# B&R Automation Studio project Nitto (part 2)

### Global.typ - Global data types
```iecst
(********************************************************************
 * COPYRIGHT -- Bernecker + Rainer
 ********************************************************************
 * File: Global.typ
 * Author: schoenefeldr
 * Created: July 06, 2012
 ********************************************************************
 * Global data types of project 120706_hp_001
 ********************************************************************)
(*======================================================================================================================================*)
(*GLOBAL OPERATING MODE DEFINITIONS*)
(*======================================================================================================================================*)
(*General operating mode of the machine*)

TYPE
	OpModeEnum_Type :
		(
		OPMODE_MANUAL := 0, (*Manual mode ("Hand")*)
		OPMODE_AUTOMATIC := 1, (*Automatic mode*)
		OPMODE_SETUP := 2, (*Automatic mode with additional functions ("Einrichten")*)
		OPMODE_SERVICE := 5 (*Service mode with direct access to hardware*)
		);
END_TYPE

(*General machine status*)

TYPE
	MachineStatusEnum_Type :
		(
		STATE_PREOPERATIONAL := 0, (*Machine not ready for operation*)
		STATE_READY_FOR_OPERATION := 1, (*Machine ready for operation*)
		STATE_AUTOMATIC := 2, (*Machine is running in operating mode automatic*)
		STATE_JOG := 3, (*Jog mode active*)
		STATE_MANUAL := 4, (*Manual operating mode*)
		STATE_FAULT := 5 (*Fault active*)
		);
END_TYPE

(*Cutting unit operating mode*)

TYPE
	OpModeCutEnum_Type :
		(
		CUT_DISABLED := 20, (*Cut unit disabled*)
		FREE_CUT := 21, (*Free cutting mode*)
		PHYSICAL_TRIGGER := 22, (*synchronous cutting mode*)
		VIRTUAL_TRIGGER := 23 (*synchronous cutting mode*)
		);
END_TYPE

(*Laaminator operating mode 17.01.14 opirational Mode*)

TYPE
	OpModeLaminatorEnum_Type :
		(
		LAMINATOR_DISABLED := 0,
		LAMINATOR_ENABLED := 1
		);
END_TYPE

(*Label dispenser operating mode*)

TYPE
	OpModeLabelDispenser_Type :
		(
		LABEL_DISP_DISABLED := 0, (*Label dispenser disabled*)
		LABEL_DISP_ENABLED := 1 (*Label dispenser enabled*)
		);
END_TYPE

(*Long cut unit operating mode*)

TYPE
	OpModeLongCutEnum_Type :
		(
		LONG_CUT_DISABLED := 10, (*Long cut enabled*)
		LONG_CUT_ENABLED := 11 (*active braking*)
		);
END_TYPE

(*Winder operating mode*)

TYPE
	OpModeWinderEnum_Type :
		(
		WIND_DISABLED := 35, (*Winder disabled*)
		WINDER := 36, (*Machine ready for operation*)
		BRAKE := 37 (*Brake functionality*)
		);
END_TYPE

(*Web tension unit operating mode*)

TYPE
	OpModeTensionEnum_Type :
		(
		WEB_TENSION_DISABLED := 5, (*Web tension control disabled*)
		WEB_TENSION_ENABLED := 6 (*Web tension control enabled*)
		);
END_TYPE

(*End module operating mode*)

TYPE
	OpModeEndModuleEnum_Type :
		(
		END_MODULE_DISABLED := 40, (*No end module selected, disable winder and belts*)
		END_MODULE_TOP_WINDER := 41, (*Select top winder*)
		END_MODULE_BOT_WINDER := 42, (*Select bottom winder*)
		END_MODULE_TANDEM_WINDER := 43, (*Select tandem winder*)
		END_MODULE_BELTS := 44 (*Select upper belt and conveyor belt*)
		);
END_TYPE

(*Markpoint operating mode*)

TYPE
	OpModeMarkpointEnum_Type :
		(
		DISABLED := 0, (*deactivated*)
		SENSOR_CONTROL := 1, (*Use sensor*)
		PERIOD_CONTROL := 2 (*use period*)
		);
	CONST_MACHINE_MODES_Type : 	STRUCT
		MANUAL : INT := 0;
		AUTOMATIC : INT := 1;
		PRODUCTION : INT := 2;
		SAFETYSTOP : INT := 7;
		RESET : INT := 8;
		EMERGENCYSTOP : INT := 9;
	END_STRUCT;
END_TYPE

(*Machine structure*)

TYPE
	Machine_Type : 	STRUCT
		Command : MachineCmd_Type;
		Safety : MachineSafe_Type;
		Data : MachineData_Type;
		Config : MachineCfg_Type;
		IO : MachineIo_Type; (*Inputs on DI9371-38A7 to DI9371-38A10*)
		Status : MachineStatus_Type;
	END_STRUCT;
	MachineCmd_Type : 	STRUCT
		StartRequestButton : BOOL; (*Start request by pressing of button*)
		StopRequestButton : BOOL; (*Stop request by pressing of button*)
		AutoStopRequestAlarm : BOOL; (*Stop request by alarm handling (automatic mode only)*)
		JogRequestButton : BOOL; (*Jog request by pressing of button*)
		UpdateRecipe : BOOL; (*Command for updating recipe parameters*)
		OpModeSet : OpModeEnum_Type; (*operating mode setpoint*)
		MasterVelocity : REAL; (*master velocity setpoint [µm/s]*)
	END_STRUCT;
	MachineSafe_Type : 	STRUCT
		RequestSTO : BOOL; (*Emergency Stop is requested (active low)*)
		RequestSLS : BOOL; (*Safe Limited Speed requested by opening safety doors (active low)*)
		ResetSafeMC : BOOL; (*Reset input of SafeMC Function Blocks*)
		ResetStartupInhibit : BOOL; (*Reset emergency functions (quit startup inhibit)*)
		ResetUserSafeMC : BOOL;
		SLSmasterVeloScaled : REAL; (*maximum master velocity command if SLS is requested due to scalings of cutting units*)
	END_STRUCT;
	MachineData_Type : 	STRUCT
		cut1 : MachineDataCut_Type; (*Derived data for cutting unit 1*)
		cut2 : MachineDataCut_Type; (*Derived data for cutting unit 2*)
		AccMaster : BOOL; (*Accelerate master axis*)
		StopMaster : BOOL; (*Decelerate master axis with machine deceleration ramp*)
		DiscreteMove : BOOL; (*Discrete move over distance or fixed number of packages*)
		VelocityIncrement : REAL; (*Increment for accelerate / decelerate master*)
	END_STRUCT;
	MachineDataCut_Type : 	STRUCT  (*Derived cuttin unit data *)
		cutPeriodLength : REAL; (*Material period corresponding to cutting cylinder perimeter [µm]*)
		scaleCutToMasterPeriod : REAL; (*Scaling factor for conversion of cutting unit into master unit*)
	END_STRUCT;
	MachineCfg_Type : 	STRUCT  (*Configuration data structure*)
		FlengeDMS : USINT; (*Configuration of Flenge DMS analogue input*)
	END_STRUCT;
	MachineStatus_Type : 	STRUCT
		initDone : BOOL; (*Initialisation complete*)
		recipeUpdating : BOOL; (*recipe updating is active*)
		recipeUpdateDone : BOOL; (*recipe update in all units completed*)
		Diam : MachineStatusDiam_Type; (*actual diameters*)
		Act : MachineStatusEnum_Type; (*actual machine status*)
		OpModeAct : OpModeEnum_Type; (*actual operating mode*)
		CalcDiam : MachineCalcDiam_Type; (*actual estimated diameter *)
		Power : BOOL; (*drives enabled*)
		ReferencedOK : BOOL; (*Combination of necessary reference conditions to start*)
		SupportSpikesOK : BOOL; (*Necessary supportspikes for tandem winders are closed*)
		mManualModeActive : BOOL;
		mAutoModeActive : BOOL;
		StartButtonBlinking : BOOL;
		StartButtonActOut : BOOL;
		WebBreakLabeler : BOOL;
		EnableMasterMove : BOOL;
	END_STRUCT;
	MachineStatusDiam_Type : 	STRUCT
		MainUnwind : REAL; (*Actual diameter Abwicklung*)
		Spend1 : REAL; (*Actual diameter Abwickler 1*)
		Spend2 : REAL; (*Actual diameter Abwickler 2*)
		Spend3 : REAL; (*Actual diameter Abwickler 3*)
		Spend4 : REAL; (*Actual diameter Abwickler 4*)
		Grid1 : REAL; (*Actual diameter Gitteraufwickler 1*)
		Grid2 : REAL; (*Actual diameter Gitteraufwickler 2*)
		Laminator1 : REAL; (*Actual diameter Laminator 1*)
		Laminator2 : REAL; (*Actual diameter Laminator 2*)
		TUnwindTop : REAL; (*Actual diameter Tandemwickler oben*)
		TUnwindBot : REAL; (*Actual diameter Tandemwickler unten*)
	END_STRUCT;
	MachineCalcDiam_Type : 	STRUCT
		MainUnwind : REAL; (*Actual estimated diameter Abwicklung*)
		TUnwindTop : REAL; (*Actual estimated diameter Tandemwickler oben*)
		TUnwindBot : REAL; (*Actual estimated diameter Tandemwickler unten*)
	END_STRUCT;
END_TYPE

(*Data types for print marks*)

TYPE
	PrintMark_Type : 	STRUCT
		Data : PrintMarkData_Type;
		ActIndex : USINT;
		MaxArrIndex : USINT;
	END_STRUCT;
	PrintMarkData_Type : 	STRUCT
		ActDiff : REAL;
		LastPos : REAL;
		AbsPos : REAL;
	END_STRUCT;
END_TYPE

(*Data types for visualisation*)

TYPE
	Visu_Type : 	STRUCT
		RelSafeOut : BOOL;
		Cmd : VisuCmd_Type;
		Status : VisuStatus_Type;
	END_STRUCT;
	VisuCmd_Type : 	STRUCT
		pageSel : VisuCmdPage_Type;
		resetError : BOOL;
		DoReference : BOOL;
		Hold : BOOL;
		StartAddPos : BOOL;
		numPkg : UDINT; (*Input for movement over a number of packages*)
		jogOverride : REAL; (*override for jogging in percent*)
		masterPos : REAL;
		masterVelo : REAL;
	END_STRUCT;
	VisuCmdPage_Type : 	STRUCT
		selPage : UINT;
		reqPage : UINT;
		actPage : UINT := 100;
		newPage : UINT;
		oldPage : UINT;
	END_STRUCT;
	VisuStatus_Type : 	STRUCT
		ActVelocity : REAL; (*Actual master speed [µm/s]*)
		ActPosition : REAL; (*Actual master position [µm]*)
	END_STRUCT;
	mAutoPunchPar_typ : 	STRUCT
		Mode : OpModeCutEnum_Type;
		TriggerIndex : USINT;
		RmWindow : REAL;
		PositionPunch : DINT;
		PositionSensor : DINT;
		CutStartPos : DINT;
		CutEndPos : DINT;
		Insetting : REAL;
		RegMarkPosition : DINT;
		MaxCorr : DINT;
	END_STRUCT;
		RmIfStatusActVal_Type : 	STRUCT  (*Structure for actual data, positions, differences etc.*)
		RmDetected : BOOL; (*A registration mark has been detected during the last movement*)
		RmShiftValid : BOOL; (*The shift value has been calculated after a valid registration mark has been detected*)
		lastValidIndex : USINT; (*Returns the last valid index of the RM data*)
		RegMark : ARRAY[0..MAX_RM_DATA_ARRAY_INDEX]OF RmActValArray_Type; (*Arrays for each registraion mark sensor*)
	END_STRUCT;
		RmActValArray_Type : 	STRUCT  (*Structure for actual data for visualisation*)
		Ident : UDINT; (*Serial number of the registration mark*)
		PIdx : USINT; (*Group index for this RM*)
		RegMarkActPos : DINT; (*Actual RM position [axis units]*)
		AbsPosition : REAL; (*Absolute position of the RM [µm]*)
		Difference : REAL; (*Difference between absolute positions [µm]*)
		SetpointError : REAL; (*Difference between RM position and setpoint [µm]*)
	END_STRUCT;
		reg_mark_typ : 	STRUCT  (*control structure*)
		Command : reg_mark_command_typ; (*command structure*)
		Parameter : reg_mark_parameter_typ; (*parameter structure*)
		Data : reg_mark_data_typ; (*data structure*)
		Status : reg_mark_status_typ; (*status structure*)
	END_STRUCT;
		reg_mark_command_typ : 	STRUCT  (*command structure*)
		StartCorrection : BOOL; (*start the correction*)
		StopCorrection : BOOL; (*stop the correction*)
		SearchTrigger : BOOL; (*search trigger manual*)
		ResetCalc : BOOL; (*reset the calculation data*)
		InitCalcData : BOOL; (*initialize the changed calculation parameters*)
		InitCaptureData : BOOL; (*initialize the changed capture parameters *)
	END_STRUCT;
	reg_mark_parameter_typ : 	STRUCT  (*parameter structure*)
		Mode : USINT; (*RM control mode, e.g. real RMs, virtual RMs etc.*)
		RegMarkAdditiveSetpoint : REAL; (*Additive cumulated RM position*)
		Capture : reg_mark_parameter_capture_typ; (*capture parameter structure*)
		Calculation : MC_RMCALC001_REF; (*ControllerParameter input structure of MC_BR_RegMarkCalc001*)
		Shift : reg_mark_parameter_shift_typ; (*shift parameter structure*)
	END_STRUCT;
	reg_mark_parameter_capture_typ : 	STRUCT  (*capture parameter structure*)
		Trigger : MC_BR_TRIGGER_REF; (*trigger input structure of MC_BR_RegMarkCapture001*)
		Product : MC_BR_PRODUCT_REF; (*product input structure of MC_BR_RegMarkCapture001*)
		WindowNegative : REAL; (*window in which the valid trigger signal can occur before the expected position*)
		WindowPositive : REAL; (*window in which the valid trigger signal can occur after the expected position*)
		DistanceToSensor : REAL; (*distance between the sensor and the cut/seal position*)
	END_STRUCT;
	reg_mark_parameter_shift_typ : 	STRUCT  (*shift parameter structure*)
		Velocity : REAL; (*maximum velocity for reaching the shift *)
		Acceleration : REAL; (*maximum acceleration for reaching the shift*)
		ApplicationDistanceRatio : REAL; (*ratio of shift application distance / product length (must be <1.0!!!)*)
	END_STRUCT;
	reg_mark_data_typ : 	STRUCT
		resetDone : BOOL; (*handshake with interface for reset command*)
		probeTriggered : BOOL; (*handshake with touchProbe*)
		actRmArrIndex : USINT; (*Write pointer index for array of RM data*)
		axisIndex : USINT; (*Index on global axis handle*)
		config : UDINT; (*configuration bits (available etc.)*)
		attrib : UDINT; (*attribute bits (reserved)*)
		rmStep : USINT; (*general registration mark control step state*)
		tpStep : USINT; (*touch probe step state*)
		lastNumOfValidTriggers : UDINT; (*Last number of valid triggers*)
		receiveParID : UINT; (*ParID of the cyclic data transfer-channel that has been automatically determined*)
		eventDelayTime : REAL; (*estimated transmission delay time [s] (unit "s" avoids division in cyclic task)*)
		eventDelayPosCompensation : REAL; (*estimated position correction for compensation of transmission delay via POWERLINK*)
	END_STRUCT;
	reg_mark_status_typ : 	STRUCT  (*status structure*)
		initDone : BOOL; (*Initialisation completed*)
		Capture : reg_mark_status_capture_typ; (*capture status structure*)
		Calculation : reg_mark_status_calc_typ; (*calculation status structure*)
		ErrorID : UINT; (*ErrorID if an function block reports an error*)
	END_STRUCT;
	reg_mark_status_capture_typ : 	STRUCT  (*capture status structure*)
		ValidTriggers : UDINT; (*number of valid triggers found by the function block*)
		MissedTriggers : UINT; (*number of missed triggers*)
		ActProbePosition : DINT; (*actual position of the last found trigger by TouchProbe*)
		ActLength : REAL; (*actual length of the last found trigger*)
		ActLengthIV : REAL; (*actual length of the interval*)
		ActPosition : REAL; (*actual position of the last found trigger*)
		LengthError : REAL; (*length error of the last interval*)
		SavePositionError : REAL; (*save variable for change detection*)
		PositionError : REAL; (*actual position error of the last found trigger*)
		SetpointError : REAL; (*Setpoint error between RM position setpoint and RM position actual value [µm]*)
		Reserve : REAL; (*Reserve*)
	END_STRUCT;
	reg_mark_status_calc_typ : 	STRUCT  (*calculation status structure*)
		ErrorID : UINT; (*ErrorID*)
		ValidCorrections : UDINT; (*number of valid calculated corrections*)
		Distance : REAL; (*calculated distance difference*)
		Shift : REAL; (*calculated shift*)
		DistanceLimiterActive : BOOL; (*shows if the calculated distance was limited to maximum*)
		ShiftLimiterActive : BOOL; (*shows if the calculated shift was limited to maximum*)
	END_STRUCT;
		RmIf_Type : 	STRUCT
		Command : RmIfCmd_Type; (*Command structure*)
		Para : RmIfPara_Type; (*Parameter structure*)
		Data : RmIfData_Type; (*General data structure*)
		Status : RmIfStatus_Type; (*Status structure*)
		Error : RmIfError_Type; (*Error data structure*)
	END_STRUCT;
	RmIfCmd_Type : 	STRUCT  (*Command structure*)
		startGeneral : BOOL; (*command for starting (depends on operating mode)*)
		stopGeneral : BOOL; (*command for starting (depends on operating mode)*)
		updatePara : BOOL; (*command for starting parameter update*)
		shadowArrayLocked : BOOL; (*command that inhibits writing to the shadow arrays*)
		clearArray1 : BOOL; (*command for clearing RM array 1*)
		clearArray2 : BOOL; (*command for clearing RM array 2*)
		reset : BOOL; (*command for reset one/all errors*)
	END_STRUCT;
	RmIfPara_Type : 	STRUCT
		axisNumber : USINT; (*axisNumber for specific commands*)
		Cut1_HomingMode : USINT; (*Tool specific homing mode for Cutting Unit 1*)
		Cut2_HomingMode : USINT; (*Tool specific homing mode for Cutting Unit 2*)
	END_STRUCT;
	RmIfData_Type : 	STRUCT  (*General data structure*)
		changeParaLatch : BOOL; (*Changing of parameters *)
		mainStep : USINT; (*main step of the registration mark control interface*)
	END_STRUCT;
	RmIfStatus_Type : 	STRUCT  (*Status structure*)
		initDone : BOOL; (*Basic interface initialisation completed*)
		rmReady : BOOL; (*registration mark task is ready for operation, may be reset during recipe loading etc.*)
		paraUpdateDone : BOOL; (*parameter update completed*)
		automaticActive : BOOL; (*status machine moves continuously, only stop allowed*)
		isMoving : BOOL; (*status machine is moving (any command)*)
		inSync : BOOL; (*status machine is in synchronized motion and "in gear"*)
		error : BOOL; (*status that at least one function block of the registration mark control has a PLCopen error*)
		ActData : ARRAY[0..MAX_RM_SENSORS_INDEX]OF RmIfStatusActVal_Type; (*Actual data, positions, differences etc.*)
	END_STRUCT;
	RmIfError_Type : 	STRUCT  (*error structure "current active" error*)
		AxisID : STRING[14]; (*axis type (Axis, Master or Slave)*)
		AxisIndex : USINT; (*index of error reporting axis (total axis index)*)
		ErrorText : ARRAY[0..4]OF STRING[79]; (*description of first active error or warning*)
		ErrorRecord : MC_ERRORRECORD_REF; (*error record information*)
		ErrorID : UDINT;
	END_STRUCT;
		Cut_Type : 	STRUCT
		MachCut : CutMachData_Type;
		CutUnitRecipe : rcp_prog_cutUnit_typ;
		rmMachineRec : rcp_machine_markpoint_typ; (*machine recipe structure*)
	END_STRUCT;
	rcp_machine_markpoint_typ : 	STRUCT
		maxRmWidth : REAL; (*maximum width of one registration mark [µm]*)
		minRmWidth : REAL; (*minimum width of one registration mark [µm], minimum < maxmum!*)
		sensorDelay : DINT; (*sensor delay [µs]*)
		sensorToolDistance : REAL; (*distance between sensor and tool [µm]*)
	END_STRUCT;
	CutMachData_Type : 	STRUCT
		Diam : REAL;
	END_STRUCT;
END_TYPE
```

### Package Logical/Libraries - Globale Bibliotheken

### Library Logical/Libraries/CSV_File (IEC, version 2.02.2)
Depends on: AsMem, AsString, FileIO, runtime, standard, sys_lib, astime

#### CSV_File.typ
```iecst
TYPE
	CSV_ListFileOption_typ : 	STRUCT
		SearchVarName : STRING[80];
		FileLenToRead : UINT;
		MaxNrLen : USINT;
		MaxNameLen : USINT;
	END_STRUCT;
	_csv_exfilelist_internal : 	STRUCT
		Step : USINT;
		DownLines : UINT;
		UpLines : UINT;
		PosFirstLine : UINT;
		FileNumOnDisk : UINT;
		FileNumAct : UINT;
		Offset : UDINT;
		TmpExtension : STRING[4];
		FileInfo : fiDIR_READ_DATA;
		i : UINT;
		result1 : DINT;
		result2 : DINT;
		OptionStruct : CSV_ListFileOption_typ;
		TmpString : ARRAY[0..50] OF USINT;
		dateandtime : DTStructure;
		status_alloc : UINT;
		pFileData : UDINT;
		FileIdent : UDINT;
		FileFound : BOOL;
		PositionFound : BOOL;
		FirstSeperatorFound : BOOL;
		SecondSeperatorFound : BOOL;
		EndPositionFound : BOOL;
		StartPositionName : UDINT;
		EndPositionName : UDINT;
		CRLF : ARRAY[0..2] OF USINT;
		InternalFileName : ARRAY[0..254] OF USINT;
		VarNameSearch : ARRAY[0..5] OF USINT;
		CompleteEntry : ARRAY[0..254] OF USINT;
	END_STRUCT;
	_csv_filelist_Internal : 	STRUCT
		MaxFileNum : UINT;
		EntriesOnDisp : USINT;
		pFileDevice : UDINT;
		pFilelist : UDINT;
		pActName : UDINT;
		pTeeList : UDINT;
		Offset : UDINT;
		MemTempOffset : UDINT;
		TempMemLng : UDINT;
		ListboxPos : UINT;
		FilePosCounter : UINT;
		FileNumAct : UINT;
		FileNumOnDisk : UINT;
		AllocStatus : UINT;
	END_STRUCT;
	_csv_init_Internal : 	STRUCT
		PV_xgetadrStatus : UINT;
		PV_ninfoStatus : UINT;
		PV_itemStatus : UINT;
		TMP_allocStatus : UINT;
		Dimension : UINT;
		ItemNrSoll : ARRAY[0..49] OF UINT;
		ItemNrIst : ARRAY[0..49] OF UINT;
		i : UINT;
		CRLF : ARRAY[0..2] OF USINT;
		Ebene : USINT;
		Step : USINT;
		FoundChar : USINT;
		Counter_Usint : USINT;
		NameCounter : USINT;
		Merker : USINT;
		MerkerArray : ARRAY[0..49] OF BOOL;
		DataLenght : UDINT;
		Datatyp : UDINT;
		PV_Adress : UDINT;
		Lenght : UDINT;
		TmpValue : UDINT;
		StartVarName : ARRAY[0..79] OF USINT;
		FullStrukturName : ARRAY[0..299] OF USINT;
		StrukturName : ARRAY[0..299] OF USINT;
		Index : ARRAY[0..6] OF USINT;
		VarItemName : ARRAY[0..299] OF USINT;
		ItemName : ARRAY[0..79] OF USINT;
		ArrayName : ARRAY[0..79] OF USINT;
		Value : ARRAY[0..79] OF USINT;
		UsintArray : ARRAY[0..79] OF USINT;
		DintTime : DINT;
		NextItemReady : BOOL;
		ArrayStructure : BOOL;
		ArrayVariable : BOOL;
		VariableCounter : UDINT;
	END_STRUCT;
	_csv_read_internal : 	STRUCT
		OnlyArray : BOOL;
		OnlyArrayInStruct : BOOL;
		DateAndTime : BOOL;
		HeaderLine : BOOL;
		DynamicVariable : BOOL;
		Step : USINT;
		NameEntered : USINT;
		ArrayStructureStarts : USINT;
		level : USINT;
		TmpDateTime : ARRAY[0..79] OF USINT;
		TmpDataTyp : ARRAY[0..79] OF USINT;
		Value : ARRAY[0..79] OF USINT;
		TmpName : ARRAY[0..149] OF USINT;
		StructName : ARRAY[0..149] OF USINT;
		DataTyp : ARRAY[0..79] OF USINT;
		DateTime : ARRAY[0..79] OF USINT;
		VarName : ARRAY[0..149] OF USINT;
		y : UINT;
		status_alloc : UINT;
		status_free : UINT;
		temp_status : UINT;
		PV_xgetadrStatus : UINT;
		PV_nInfoStatus : UINT;
		PVdata_typ : UDINT;
		datatyp_len : UDINT;
		dimension : UINT;
		j : UDINT;
		i : UDINT;
		FileIdent : UDINT;
		pFileData : UDINT;
		Offset : UDINT;
		OffsetOld : UDINT;
		CharPerCyclic : UDINT;
		SpacesCounter : UDINT;
		Merker : UDINT;
		SpacesLastRow : UDINT;
		nextPV : UDINT;
		Counter : UDINT;
		PV_Adress : UDINT;
		data_len : UDINT;
		FileName : STRING[80];
		Path : STRING[80];
		DateTimeStruct : DTStructure;
		Separator : USINT;
	END_STRUCT;
	_csv_search_internal : 	STRUCT
		PV_xgetadrStatus : UINT;
		PV_ninfoStatus : UINT;
		PV_itemStatus : UINT;
		TMP_allocStatus : UINT;
		Dimension : UINT;
		ItemNrSoll : ARRAY[0..49] OF UINT;
		ItemNrIst : ARRAY[0..49] OF UINT;
		i : UINT;
		y : UINT;
		FullStrukturName : ARRAY[0..299] OF USINT;
		StrukturName : ARRAY[0..299] OF USINT;
		ArrayName : ARRAY[0..79] OF USINT;
		UsintArray : ARRAY[0..79] OF USINT;
		CRLF : ARRAY[0..2] OF USINT;
		Separator : ARRAY[0..1] OF USINT;
		Ebene : USINT;
		Step : USINT;
		NameCounter : USINT;
		FoundChar : USINT;
		Counter_Usint : USINT;
		Merker : USINT;
		MerkerArray : ARRAY[0..49] OF BOOL;
		DataLenght : UDINT;
		Datatyp : UDINT;
		PV_Adress : UDINT;
		Offset : UDINT;
		TmpValue : UDINT;
		Lenght : UDINT;
		Date_and_Time : DATE_AND_TIME;
		DintTime : DINT;
		Index : ARRAY[0..6] OF USINT;
		StartVarName : ARRAY[0..79] OF USINT;
		VarItemName : ARRAY[0..299] OF USINT;
		ItemName : ARRAY[0..79] OF USINT;
		Value : ARRAY[0..79] OF USINT;
		NextItemReady : BOOL;
		ArrayStructure : BOOL;
		ArrayVariable : BOOL;
		VariableCounter : UDINT;
	END_STRUCT;
END_TYPE
```

#### CSV_File.var
```iecst
VAR CONSTANT
	ARRAY_TO_LESS	:UINT	:=5003;
	DATATYP_ERROR	:UINT	:=5007;
	ERRF_NO_ERROR	:UINT	:=0;
	ERROR_CHECKFILEBUFFER_TOO_SMALL	:UINT	:=5013;
	ERROR_ENABLE_NOT_SET	:UINT	:=5017;
	ERROR_INPUT_POINTER_ERR	:UINT	:=5018;
	ERROR_NUM_OF_STRUCT_MISMATCH	:UINT	:=5015;
	ERROR_SIZE_MISMATCH	:UINT	:=5016;
	ERROR_STRUCTNAME_TOO_LONG	:UINT	:=5010;
	ERROR_STRUCT_NAMES	:UINT	:=5006;
	ERROR_VERSION_MISMATCH	:UINT	:=5014;
	ERROR_WRONG_SEPARATOR	:UINT	:=5012;
	ERROR_ZERO_POINTER_FILE	:UINT	:=5019;
	ERR_NO_MEM_ALLOC	:UINT	:=5000;
	ERR_PV_ADRESS	:UINT	:=5008;
	ERR_ZERO_POINTER_DEVICE	:UINT	:=5009;
	ERR_ZERO_POINTER_OPTION	:UINT	:=5011;
	EXECUTION_BUSY	:UINT	:=0;
	FILE_CREATE	:USINT	:=0;
	FILE_CREATE_WITHOUT_MEM_CHECK	:USINT	:=2;
	FILE_FOUND	:UINT	:=1;
	FILE_NOT_FOUND	:UINT	:=0;
	FILE_OW	:USINT	:=1;
	FILE_OW_WITHOUT_MEM_CHECK	:USINT	:=3;
	FOCUSPOS_OUT_OF_LISTBOX	:UINT	:=5005;
	FiJOB_CREATE_FILE_LIST	:USINT	:=2;
	FiJOB_LIST_DOWN	:USINT	:=6;
	FiJOB_LIST_PG_DOWN	:USINT	:=4;
	FiJOB_LIST_PG_UP	:USINT	:=3;
	FiJOB_LIST_UP	:USINT	:=5;
	FiJOB_SET_FOCUS	:USINT	:=7;
	HEADER	:BOOL	:=TRUE;
	INVALID_CHARACTER	:UINT	:=5004;
	MAX_NAMELENGHT_TO_LONG	:UINT	:=5002;
	MAX_VAR_NAME_LENGHT	:UINT	:=40;
	NO_FILENAME	:UINT	:=5001;
	NO_HEADER	:BOOL	:=FALSE;
END_VAR
```

#### CSV_File.fun
```iecst
FUNCTION_BLOCK CSV_CheckFile
	VAR_INPUT
		enable : BOOL;
		pFileName : UDINT;
		pDevice : UDINT;
		pStructSizes : UDINT;
		NumOfStruct : USINT;
		pVersion : UDINT;
		pFileBuffer : UDINT;
		FileBufferSize : UDINT;
	END_VAR
	VAR_OUTPUT
		status : UINT;
		fileError : UINT;
	END_VAR
	VAR
		statusInternal : UINT;
		fileVersionStr : STRING[255];
		cntSizesFound : USINT;
		ixCmp : USINT;
		pSize : REFERENCE TO UDINT;
		SizesFound : ARRAY[0..254] OF UDINT;
		fileOffset : UDINT;
		sizeSignificationStr : STRING[255];
		lineBuf : STRING[255];
		versionFound : BOOL;
		maxLenLine : UINT;
		ixLine : UDINT;
		ixLineMax : UDINT;
		lineCnt : UDINT;
		FClose : FileClose;
		fileIdent : UDINT;
		pChar : REFERENCE TO USINT;
		FOpen : FileOpen;
		FRead : FileRead;
		verSignificationStr : STRING[255];
		R_TRIG_0 : R_TRIG;
		fileCheckStep : UINT;
		CharPerCyclic : USINT;
	END_VAR
END_FUNCTION_BLOCK

FUNCTION_BLOCK CSV_InitCheckFile
	VAR_INPUT
		enable : BOOL;
		MemCounter : UDINT;
	END_VAR
	VAR_OUTPUT
		status : UINT;
		pFileBuffer : UDINT;
		FileBufferSize : UDINT;
	END_VAR
	VAR
		AsMemPartAlloc_0 : AsMemPartAlloc;
		AsMemPartCreate_0 : AsMemPartCreate;
	END_VAR
END_FUNCTION_BLOCK

FUNCTION_BLOCK CSV_Search
	VAR_INPUT
		pStructName : UDINT;
		NumOfStructs : USINT;
		pStructMem : UDINT;
		MemLen : UDINT;
		Options : UDINT;
		FullNameLenght : BOOL;
		FileHeader : BOOL;
		Separator : USINT;
		pMaschineNo : UDINT;
		pComment : UDINT;
		pVersion : UDINT;
	END_VAR
	VAR_OUTPUT
		status : UINT;
		ErrorName : USINT;
		FileLen : UDINT;
	END_VAR
	VAR
		Internal : _csv_search_internal;
		zzDTGetTime00000 : DTGetTime;
		SearchChar : REFERENCE TO USINT;
		Dyn_Bool : REFERENCE TO BOOL;
		Dyn_Usint : REFERENCE TO USINT;
		Dyn_Sint : REFERENCE TO SINT;
		Dyn_Uint : REFERENCE TO UINT;
		Dyn_Int : REFERENCE TO INT;
		Dyn_Udint : REFERENCE TO UDINT;
		Dyn_Dint : REFERENCE TO DINT;
		Dyn_Real : REFERENCE TO REAL;
		Dyn_LReal : REFERENCE TO LREAL;
		Dyn_Date_and_Time : REFERENCE TO DATE_AND_TIME;
		Dyn_Time : REFERENCE TO TIME;
		OnlyOneVar : BOOL;
	END_VAR
END_FUNCTION_BLOCK

FUNCTION_BLOCK CSV_Init
	VAR_INPUT
		pStructName : UDINT;
		NumOfStructs : USINT;
		FullNameLenght : BOOL;
		Options : UDINT;
	END_VAR
	VAR_OUTPUT
		status : UINT;
		ErrorName : USINT;
		pStructMem : UDINT;
		MemCounter : UDINT;
	END_VAR
	VAR
		Internal : _csv_init_Internal;
		SearchChar : REFERENCE TO USINT;
		Dyn_Usint : REFERENCE TO USINT;
		Dyn_Sint : REFERENCE TO SINT;
		Dyn_Int : REFERENCE TO INT;
		Dyn_Dint : REFERENCE TO DINT;
		Dyn_Uint : REFERENCE TO UINT;
		Dyn_Udint : REFERENCE TO UDINT;
		Dyn_Real : REFERENCE TO REAL;
		Dyn_LReal : REFERENCE TO LREAL;
		Dyn_Date_and_Time : REFERENCE TO DATE_AND_TIME;
		Dyn_Time : REFERENCE TO TIME;
		OnlyOneVar : BOOL;
	END_VAR
END_FUNCTION_BLOCK

FUNCTION_BLOCK CSV_ListFile
	VAR_INPUT
		pStringArray : UDINT;
		SizeStringArray : UDINT;
		ArrayNum : UINT;
		NumListboxLines : UINT;
		pFileDevice : UDINT;
		pPath : UDINT;
		MaxNameLenght : USINT;
		SetFocusPos : UINT;
		command : USINT;
	END_VAR
	VAR_OUTPUT
		status : UINT;
		CSV_FileNum : UINT;
		ListboxFocusPos : UINT;
		ScrollUp : BOOL;
		ScrollDown : BOOL;
	END_VAR
	VAR
		DirRead_01 : DirRead;
		DirInfo_01 : DirInfo;
		TmpString : ARRAY[0..50] OF USINT;
		Step : USINT;
		i : UINT;
		TmpExtension : STRING[4];
		FileInfo : fiDIR_READ_DATA;
		result1 : DINT;
		result2 : DINT;
		FileNumAct : UINT;
		FileNumOnDisk : UINT;
		Offset : UDINT;
		dateandtime : DTStructure;
		UpLines : UINT;
		DownLines : UINT;
		PosFirstLine : UINT;
		xFileNameWithDate : BOOL; (*set to 1 if the date and time of file is needed*)
	END_VAR
END_FUNCTION_BLOCK

FUNCTION_BLOCK SearchFileName
	VAR_INPUT
		pFileName : UDINT;
		pDevice : UDINT;
	END_VAR
	VAR_OUTPUT
		status : UINT;
	END_VAR
	VAR
		step : USINT;
		FileName : STRING[40];
		i : USINT;
		FileOpen_01 : FileOpen;
		FileClose_01 : FileClose;
		SearchChar : REFERENCE TO USINT;
	END_VAR
END_FUNCTION_BLOCK

FUNCTION_BLOCK CSV_ReadFile
	VAR_INPUT
		pFileName : UDINT;
		pDevice : UDINT;
		pPath : UDINT;
		No_DatatypControl : BOOL;
		Separator : USINT;
		IgnoreError : BOOL;
		Options : UDINT;
	END_VAR
	VAR_OUTPUT
		status : UINT;
		LineCnt : UDINT;
		VarCnt : UDINT;
		ErrorLine : UDINT;
		ErrorNumber : UINT;
		ErrorCnt : UDINT;
	END_VAR
	VAR
		FileOpen_CSV : FileOpen;
		FileRead_CSV : FileRead;
		FileClose_CSV : FileClose;
		Internal : _csv_read_internal;
		Dyn_Usint : REFERENCE TO USINT;
		SearchChar : REFERENCE TO USINT;
		Dyn_Bool : REFERENCE TO BOOL;
		Dyn_Sint : REFERENCE TO SINT;
		Dyn_Uint : REFERENCE TO UINT;
		Dyn_Int : REFERENCE TO INT;
		Dyn_Udint : REFERENCE TO UDINT;
		Dyn_Dint : REFERENCE TO DINT;
		Dyn_String : REFERENCE TO STRING[255];
		Dyn_Real : REFERENCE TO REAL;
		Dyn_LReal : REFERENCE TO LREAL;
		Dyn_Date_and_Time : REFERENCE TO DATE_AND_TIME;
		Dyn_Time : REFERENCE TO TIME;
		Part : BOOL;
		TestUsint : USINT;
		temp_status : UINT;
	END_VAR
END_FUNCTION_BLOCK

FUNCTION_BLOCK ExListFile
	VAR_INPUT
		pStringArray : UDINT;
		SizeStringArray : UDINT;
		NumListboxLines : UINT;
		ArrayNum : UINT;
		pFileDevice : UDINT;
		MaxNameLenght : USINT;
		SetFocusPos : UINT;
		command : USINT;
		pOptions : UDINT;
	END_VAR
	VAR_OUTPUT
		status : UINT;
		CSV_FileNum : UINT;
		ListboxFocusPos : UINT;
		ScrollUp : BOOL;
		ScrollDown : BOOL;
	END_VAR
	VAR
		Internal : _csv_exfilelist_internal;
		DirInfo_CSV : DirInfo;
		DirRead_CSV : DirRead;
		FileOpen_CSV : FileOpen;
		FileRead_CSV : FileRead;
		FileClose_CSV : FileClose;
		DynUsint : REFERENCE TO USINT;
	END_VAR
END_FUNCTION_BLOCK

FUNCTION_BLOCK CSV_WriteFile
	VAR_INPUT
		pFileName : UDINT;
		pDevice : UDINT;
		pPath : UDINT;
		pStructMem : UDINT;
		MemLen : UDINT;
		Mode : USINT;
	END_VAR
	VAR_OUTPUT
		status : UINT;
	END_VAR
	VAR
		Step : USINT;
		FileCreate_CSV : FileCreate;
		FileWrite_CSV : FileWrite;
		FileDelete_CSV : FileDelete;
		FileClose_CSV : FileClose;
		FileName : STRING[80];
		i : USINT;
		Dyn_Usint : REFERENCE TO USINT;
		DevMemInfo_CSV : DevMemInfo;
		Path : STRING[100];
		DirInfo_CSV : DirInfo;
	END_VAR
END_FUNCTION_BLOCK

FUNCTION CSV_AtoDouble : LREAL (*Converts an ASCII-String to a LREAL-Value*)
	VAR_INPUT
		pString : UDINT; (*Adress of to String which has to be converted*)
	END_VAR
	VAR
		intStrLeng : UINT;
		tempString : USINT;
		negativeValue : BOOL;
		startIndexIntPart : UINT;
		i : UINT;
		lRealIntegerPart : LREAL;
		startIndexDecPart : UINT;
		decimalPlaces : BOOL;
		tempInt : DINT;
		lRealDecimalPart : LREAL;
		anzDecimalPlaces : UINT;
		anzExponent : DINT;
		positivExponent : BOOL;
	END_VAR
END_FUNCTION

FUNCTION CSV_DoubleToA : UINT (*Converts a LREAL-Value to an ASCII-String*)
	VAR_INPUT
		lRealValue : LREAL;
		pString : UDINT;
	END_VAR
	VAR
		tempLREALvalue : LREAL;
		intStringLen : UINT;
		tempInt : DINT;
		negativeValue : BOOL;
		i : DINT;
		exponent : DINT;
		IntPartLReal : DINT;
		DecPartLReal : ARRAY[0..16] OF DINT;
		tempString : STRING[20];
		firstEntry : BOOL;
		tempDecString : STRING[20];
	END_VAR
END_FUNCTION
```

#### CSV_CheckFile.ab
```automation-basic
FUNCTION_BLOCK CSV_CheckFile
(********************************************************************
 * COPYRIGHT -- Bernecker + Rainer Industrie Elektronik GmbH
 ********************************************************************
 * Library: CSV_File
 * File: CSV_CheckFile.ab
 * Author: kreidlm
 * Created: November 29, 2006
 ********************************************************************
 * Implementation of library CSV_File
 ********************************************************************)

CharPerCyclic = CharPerCyclic

R_TRIG_0.CLK = enable
R_TRIG_0 FUB R_TRIG()

select fileCheckStep of
	;##########################################################################################
    state WAIT
	;##########################################################################################

        when (R_TRIG_0.CLK = 1) and ( (pFileName = 0) or (pDevice = 0) or (pStructSizes = 0) or (pVersion = 0) or (pFileBuffer = 0) ) do
            status = ERROR_INPUT_POINTER_ERR;
       	next WAIT

        when (R_TRIG_0.CLK = 1) do
            status = 65535
            statusInternal = 0
            fileError = 0
            lineCnt = 0
            maxLenLine = SIZEOF(lineBuf)-1
            versionFound = 0
            cntSizesFound = 0
            memset(adr(SizesFound), 0, SIZEOF(SizesFound))
            strcpy(adr(verSignificationStr),"// V")
            strcpy(adr(sizeSignificationStr), "// Structure Size: ")
            strcpy(adr(fileVersionStr), "")
        next FOPEN

	;##########################################################################################
    state FOPEN
	;##########################################################################################
    	FOpen.enable = 1
        FOpen.pDevice  = pDevice
        FOpen.pFile = pFileName
        FOpen.mode = 2

        FOpen FUB FileOpen()
        fileIdent = FOpen.ident
        statusInternal = FOpen.status

        when (statusInternal = 0) and (FOpen.filelen < FileBufferSize) do
            memset(pFileBuffer, 0 , FileBufferSize)
            pChar access (pFileBuffer+FOpen.filelen)
            pChar = 0 (* Terminierung ans Ende des Filebuffers*)
            status = 65535
        next FREAD
        (* File zu gross für Buffer *)
        when (statusInternal = 0) and (FOpen.filelen >= FileBufferSize) do
        	statusInternal = ERROR_CHECKFILEBUFFER_TOO_SMALL
            status = statusInternal
        next WAIT
        when ((statusInternal <> 0) and (statusInternal <> 65535)) do
            if (statusInternal = fiERR_SYSTEM) then
                fileError = FileIoGetSysError()
            endif
            status = statusInternal
        next WAIT

	;##########################################################################################
    state FREAD
	;##########################################################################################
         FRead.enable = 1
         FRead.ident = fileIdent
         FRead.offset = 0
         FRead.pDest = pFileBuffer
         FRead.len = FOpen.filelen

         FRead FUB FileRead()
         statusInternal = FRead.status

         when (statusInternal = 0) do
            loop fileOffset = 0 to (FOpen.filelen-1) do
                pChar access (pFileBuffer+fileOffset)
                if (pChar = 10) then (* LF *)
            	    pChar = 0 (* durch Terminator ersetzen *)
                    lineCnt = lineCnt + 1
                endif
   	        endloop
            fileOffset = pFileBuffer
            status = 65535
         next FCLOSE
         when ((statusInternal <> 0) and (statusInternal <> 65535)) do
            if (statusInternal = fiERR_SYSTEM) then
                fileError = FileIoGetSysError()
            endif
            status = statusInternal
         next WAIT

	;##########################################################################################
	state FCLOSE
	;##########################################################################################
    	FClose.enable = 1
        FClose.ident = fileIdent

        FClose FUB FileClose()
        statusInternal = FClose.status

        when (statusInternal = 0) do
        	status = 65535
        next FCHECK
        when ((statusInternal <> 0) and (statusInternal <> 65535)) do
            if (statusInternal = fiERR_SYSTEM) then
                fileError = FileIoGetSysError()
            endif
            status = statusInternal
        next WAIT

	;##########################################################################################
    state FCHECK
	;##########################################################################################
        when (1=1) do
            if (lineCnt > 0) then
                ixLineMax = lineCnt - 1
            else
            	ixLineMax = 0
            endif
            ;Filebuffer parsen
            loop ixLine = 0 to ixLineMax do
                if (strlen(fileOffset) <= maxLenLine ) then
                    strcpy(adr(lineBuf), fileOffset)
                    if ((FIND(lineBuf, verSignificationStr) = 1) and (versionFound = 0)) then
                        fileVersionStr = MID(lineBuf, strlen(pVersion), strlen(adr(verSignificationStr)))
                        versionFound = 1
                    endif
                    if ((FIND(lineBuf, sizeSignificationStr) = 1) and (cntSizesFound < NumOfStruct)) then
                        SizesFound[cntSizesFound] = atoi(adr(lineBuf) + strlen(adr(sizeSignificationStr)))
                        cntSizesFound = cntSizesFound + 1
                    endif
                endif
                fileOffset = fileOffset + strlen(fileOffset) + 1
            endloop
            ;Auswertung
            if (strcmp(adr(fileVersionStr), pVersion) <> 0) then
                statusInternal = ERROR_VERSION_MISMATCH
            endif
            if (cntSizesFound <> NumOfStruct) then
        	    statusInternal = ERROR_NUM_OF_STRUCT_MISMATCH
            endif
       	    if (NumOfStruct > 0) then
                loop ixCmp = 0 to (NumOfStruct-1) do
                    pSize access (pStructSizes + ixCmp*SIZEOF(SizesFound[0]))
                    if (SizesFound[ixCmp] <> pSize) then
                        statusInternal = ERROR_SIZE_MISMATCH
                    endif
                    exitif (statusInternal = ERROR_SIZE_MISMATCH)
                endloop
            else
                statusInternal = ERROR_NUM_OF_STRUCT_MISMATCH
            endif
            status = statusInternal
      	next WAIT

endselect
END_FUNCTION_BLOCK
```

#### CSV_InitCheckFile.ab
```automation-basic
FUNCTION_BLOCK CSV_InitCheckFile
(********************************************************************
 * COPYRIGHT -- Bernecker + Rainer Industrie Elektronik GmbH
 ********************************************************************
 * Library: CSV_File
 * File: CSV_InitCheckFile
 * Author: kreidlm
 * Created: November 28, 2006
 ********************************************************************
 * Implementation of library CSV_File
 ********************************************************************)

if (enable = 1) then
    AsMemPartCreate_0.enable = 1
    AsMemPartCreate_0.len = MemCounter + 128 (* + Overhead und Reserve *)
    AsMemPartCreate_0 FUB AsMemPartCreate()
    if (AsMemPartCreate_0.status = 0) then
        AsMemPartAlloc_0.enable = 1
        AsMemPartAlloc_0.ident = AsMemPartCreate_0.ident
        AsMemPartAlloc_0.len = MemCounter
        AsMemPartAlloc_0 FUB AsMemPartAlloc()
        status = AsMemPartAlloc_0.status
        pFileBuffer = AsMemPartAlloc_0.mem
        FileBufferSize =  AsMemPartAlloc_0.len
    else
    	status = AsMemPartCreate_0.status
    endif
 else
 	status = ERROR_ENABLE_NOT_SET
 endif

END_FUNCTION_BLOCK
```
